FUNCTION_BLOCK FC_ProcedureFacade (* Fixed procedure boundary; unavailable until composition is installed; never invents completion *)
  (* Standard: 61499-2 *)
  (* Version 2.0, 2026-09-27, Project contributors, Filling cell reference model *)
  PACKAGE fillingcell;
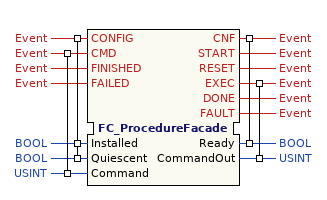
  EVENT_INPUT
    CONFIG WITH Installed, Quiescent;
    CMD WITH Command;
    FINISHED;
    FAILED;
  END_EVENT
  EVENT_OUTPUT
    CNF WITH Ready;
    START;
    RESET;
    EXEC WITH CommandOut;
    DONE;
    FAULT;
  END_EVENT
  VAR_INPUT
    Installed : BOOL;
    Quiescent : BOOL;
    Command : USINT;
  END_VAR
  VAR_OUTPUT
    Ready : BOOL;
    CommandOut : USINT;
  END_VAR
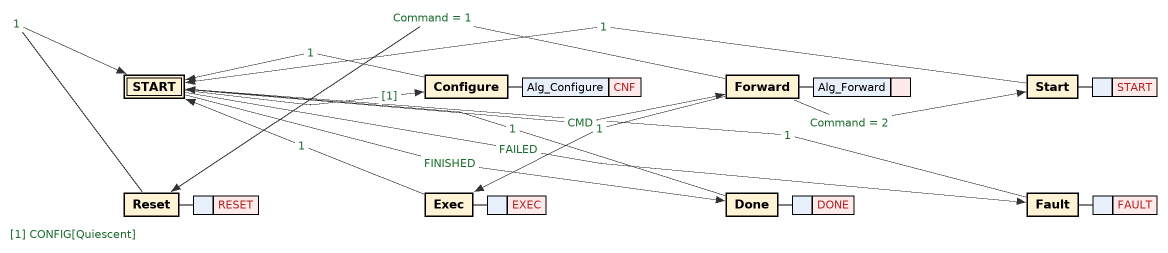
  EC_STATES
    START;
    Configure : Alg_Configure -> CNF;
    Forward : Alg_Forward;
    Start : -> START;
    Reset : -> RESET;
    Exec : -> EXEC;
    Done : -> DONE;
    Fault : -> FAULT;
  END_STATES
  EC_TRANSITIONS
    Forward TO Start := Command = 2;
    Forward TO Reset := Command = 1;
    Forward TO Exec := 1;
    Start TO START := 1;
    Reset TO START := 1;
    Exec TO START := 1;
    START TO Configure := CONFIG[Quiescent];
    Configure TO START := 1;
    START TO Forward := CMD;
    START TO Done := FINISHED;
    Done TO START := 1;
    START TO Fault := FAILED;
    Fault TO START := 1;
  END_TRANSITIONS
  ALGORITHM Alg_Configure IN ST:
Ready := Installed;
  END_ALGORITHM
  ALGORITHM Alg_Forward IN ST:
CommandOut := Command;
  END_ALGORITHM
END_FUNCTION_BLOCK
